Staubli VAL3: Form_Patten.pgx

public program Form_Patten(string x_sTitle, string& x_sLeftList[], string& x_sBottomList[])
  local num l_nIndex
begin
  //****************************************************************
  //***************************************************************
  //函数名称：pagePatten1
  //用途：  用于图形显示
  //创建日期：2013.02.18
  //作者：
  //联系方式：
  //备注：
  //版本修改说明：
  //图形类型
  //                   100%
  //=========标题================
  //
  //F1->文字1
  //F2->文字2
  //F3->文字3
  //F4->文字4
  //F5->文字5
  //F6->文字6
  //F7->文字7


  //文字  文字  文字 文字 文字 文字 文字 文字
  //****************************************************************
  //*****************************************************************



  cls()

  title(x_sTitle)


    //左边标记

    call Control_Left(x_sLeftList)
    //底部标记
    call Control_Bottom(x_sBottomList)


end
